(* PLC project Unnamed, Unknown Unnamed 1 *)
(* stored: creationDateTime 2023-03-30T12:57:47, modificationDateTime 2023-05-02T08:31:03 *)

PROGRAM program0
  VAR
    Recieve_Signal AT %IX0.0 : BOOL;
    LED AT %Q0.0 : BOOL;
  END_VAR

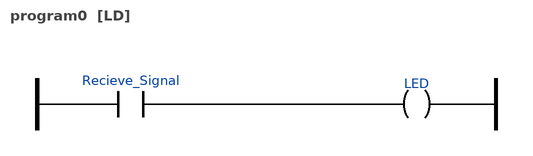
(* LD diagram, written out as Structured Text *)
LED := Recieve_Signal;
END_PROGRAM

CONFIGURATION Config0
  RESOURCE Res0 ON PLC
    TASK task0(INTERVAL := T#20ms, PRIORITY := 0);
    PROGRAM instance0 WITH task0 : program0;
  END_RESOURCE
END_CONFIGURATION
